(* PLC project  *)

CONFIGURATION DO_
END_CONFIGURATION
